{attribute 'qualified_only'}
VAR_GLOBAL
END_VAR

(* stored: Version 1.1.0.1, ProductVersion 3.1.4022.18
   GVL IN_GLV: Id {ade190a6-b1a2-4f1a-9800-79129591440f} *)
